Fanuc KAREL source: kt00580.KL

-- PROVISIONAL review KL for V770-1; original PC SHA256 021f7d5df4531234110884ed15bad4535a0e2ca06aa6f8e8ee92d7942698f9f1
-- Incomplete behavior may be omitted. Consult companion uncertainty JSON. Do not deploy.
PROGRAM KT00580
%NOLOCKGROUP
VAR
  I2 : INTEGER
-- UNRESOLVED_DECL V1 type=000013
-- UNRESOLVED_DECL OUT type=000013
BEGIN
  -- UNRESOLVED_PC offsets 5-20; opcodes 2E,22,32,35
  -- UNRESOLVED_PC offsets 25-36; opcodes 2E,23
  -- UNRESOLVED_PC offsets 41-63; opcodes 49,21,8D,4A
  -- UNRESOLVED_PC offsets 68-72; opcodes 7F
END KT00580
